Omron CX-Programmer project NewProject (CX-Programmer 9.75)

# PLC NewPLC1: CP1L M

## Global symbols (name address type ; comment)
0.00 BOOL  ; S3
0.01 BOOL  ; S4
0.02 BOOL  ; S2
0.03 BOOL  ; S1
100.00 BOOL  ; Y1_14
100.01 BOOL  ; Y2_12
100.02 BOOL  ; Y3_14
100.03 BOOL  ; Y4_12

## Program NewProgram1 (cyclic task 0)

### Section Section1

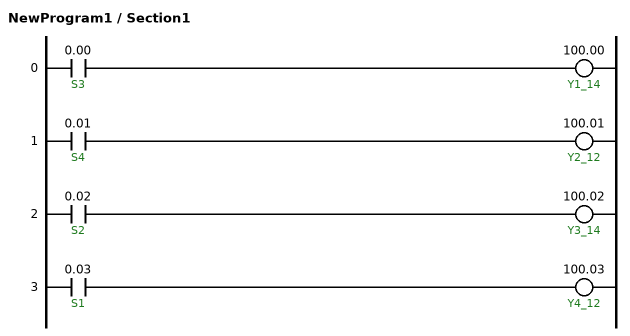
; rung 0
LD 0.00  ; S3
OUT 100.00  ; Y1_14
; rung 1
LD 0.01  ; S4
OUT 100.01  ; Y2_12
; rung 2
LD 0.02  ; S2
OUT 100.02  ; Y3_14
; rung 3
LD 0.03  ; S1
OUT 100.03  ; Y4_12

### Section END
; rung 0
END(001)